// TIA Portal project "Automatic Washing Machine" (V17)
// Automatic Washing Machine
// When Start button is pressed, it starts filling water for 10 sec, then Agitate for 30 sec, then Drain the water for 5 sec, spin the drum for 10 sec and then Buzzer will be ON for 10 sec.

(* hardware
DEVICE "S7-1200 station_1"  S7-1200 Station
   slot 0: "Rack_0"  S7-1200 Rack  Rack  V1.0
   slot 1: "PLC_1"  CPU 1211C AC/DC/Rly  6ES7 211-1BE40-0XB0  V4.5
*)

// ===== PLC "PLC_1"  CPU 1211C AC/DC/Rly =====

VAR_GLOBAL   // PLC tag table "Default tag table"
   "Start button" AT %I0.0 : Bool;
   "Fill valve" AT %Q0.0 : Bool;
   "Agitator motor" AT %Q0.1 : Bool;
   "Drain valve/pump" AT %Q0.2 : Bool;
   "Spin motor" AT %Q0.3 : Bool;
   "Buzzer" AT %Q0.4 : Bool;
   "Washmachine Program" AT %M0.0 : Bool;
END_VAR

// folder: System blocks/Program resources

DATA_BLOCK "IEC_Timer_0_DB"   // DB1
{ S7_Optimized_Access := 'TRUE' }
AUTHOR : Simatic
FAMILY : IEC
NAME : IEC_TMR
VERSION : 1.0
// stored: InstanceOfName IEC_TIMER
"IEC_TIMER"
BEGIN
END_DATA_BLOCK

DATA_BLOCK "IEC_Timer_0_DB_1"   // DB2
{ S7_Optimized_Access := 'TRUE' }
AUTHOR : Simatic
FAMILY : IEC
NAME : IEC_TMR
VERSION : 1.0
// stored: InstanceOfName IEC_TIMER
"IEC_TIMER"
BEGIN
END_DATA_BLOCK

DATA_BLOCK "IEC_Timer_0_DB_2"   // DB3
{ S7_Optimized_Access := 'TRUE' }
AUTHOR : Simatic
FAMILY : IEC
NAME : IEC_TMR
VERSION : 1.0
// stored: InstanceOfName IEC_TIMER
"IEC_TIMER"
BEGIN
END_DATA_BLOCK

DATA_BLOCK "IEC_Timer_0_DB_3"   // DB4
{ S7_Optimized_Access := 'TRUE' }
AUTHOR : Simatic
FAMILY : IEC
NAME : IEC_TMR
VERSION : 1.0
// stored: InstanceOfName IEC_TIMER
"IEC_TIMER"
BEGIN
END_DATA_BLOCK

DATA_BLOCK "IEC_Timer_0_DB_4"   // DB5
{ S7_Optimized_Access := 'TRUE' }
AUTHOR : Simatic
FAMILY : IEC
NAME : IEC_TMR
VERSION : 1.0
// stored: InstanceOfName IEC_TIMER
"IEC_TIMER"
BEGIN
END_DATA_BLOCK

// folder: (top level)

ORGANIZATION_BLOCK "Main"   // OB1, LAD, ProgramCycle
TITLE = "Main Program Sweep (Cycle)"
{ S7_Optimized_Access := 'TRUE' }
VERSION : 0.1
   VAR_INPUT
      Initial_Call : Bool;   // Initial call of this OB
      Remanence : Bool;   // =True, if remanent data are available
   END_VAR
BEGIN

REGION Network 1
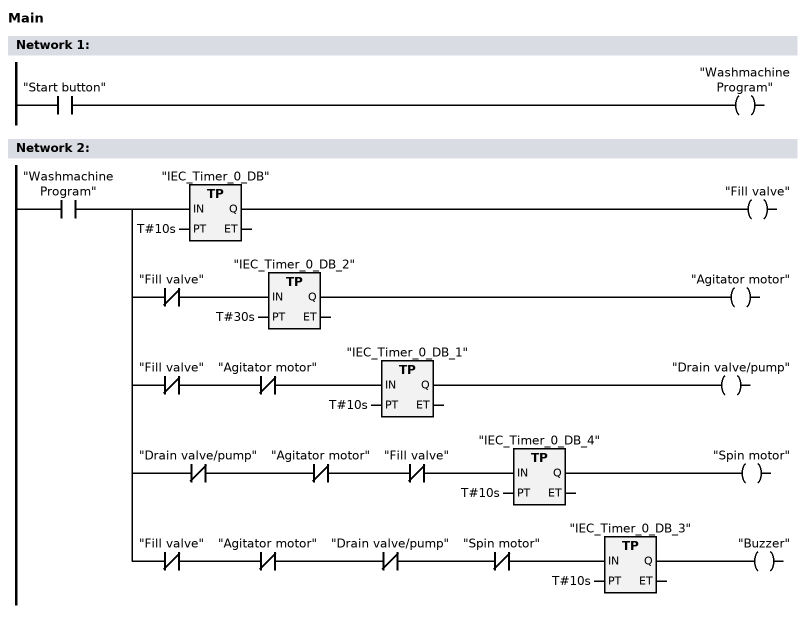
   RUNG wire#powerrail
      Contact( "Start button" )
      Coil( "Washmachine Program" )
   END_RUNG
   // the same network as SCL:
   "Washmachine Program" := "Start button";
END_REGION

REGION Network 2
   "IEC_Timer_0_DB".TP(IN := "Washmachine Program", PT := T#10s);
   "Fill valve" := "IEC_Timer_0_DB".Q;
   "IEC_Timer_0_DB_2".TP(IN := "Washmachine Program" AND NOT "Fill valve", PT := T#30s);
   "Agitator motor" := "IEC_Timer_0_DB_2".Q;
   "IEC_Timer_0_DB_1".TP(IN := "Washmachine Program" AND NOT "Fill valve" AND NOT "Agitator motor", PT := T#10s);
   "Drain valve/pump" := "IEC_Timer_0_DB_1".Q;
   "IEC_Timer_0_DB_4".TP(IN := "Washmachine Program" AND NOT "Drain valve/pump" AND NOT "Agitator motor" AND NOT "Fill valve",
                         PT := T#10s);
   "Spin motor" := "IEC_Timer_0_DB_4".Q;
   "IEC_Timer_0_DB_3".TP(IN := "Washmachine Program" AND NOT "Fill valve" AND NOT "Agitator motor" AND NOT "Drain valve/pump" AND NOT "Spin motor",
                         PT := T#10s);
   "Buzzer" := "IEC_Timer_0_DB_3".Q;
END_REGION
END_ORGANIZATION_BLOCK